// TwinCAT 3 PLC project shelf
// Title: Shelf
// Company: Stefan Lehmann
// ProjectVersion: 0.0.1
// ProgramVersion: 3.1.4026.14
// libraries:
//   Shelf, * (Stefan Lehmann)
//   Tc2_System, * (Beckhoff Automation GmbH)
//   Tc2_Utilities, * (Beckhoff Automation GmbH)
//   Tc3_Module, * (Beckhoff Automation GmbH)
// project tree:
//   / ClassDiagram.TcCD (not stored), PlcTask.TcTTO
//   classes/ FifoBuffer.TcPOU, FlexiBuffer.TcPOU, Part.TcPOU, Shelf.TcPOU, ShelfElement.TcPOU
//   enums/ MainState.TcDUT, TestFlexiBufferState.TcDUT
//   interfaces/ IPart.TcIO, IShelf.TcIO, IShelfElement.TcIO
//   programs/ main.TcPOU
//   programs/tests/ testFlexiBuffer.TcPOU, testShelf.TcPOU
// real-time tasks:
//   TASK PlcTask: cycle T#10ms, priority 1, ADS port 350
//   TASK Standard: cycle T#10ms, priority 20, ADS port 351

CONFIGURATION shelf
    RESOURCE PLC ON TwinCAT3
        TASK PlcTask(INTERVAL := T#10ms, PRIORITY := 1);
        PROGRAM main WITH PlcTask : main;
    END_RESOURCE
END_CONFIGURATION

// ---- enums/MainState.TcDUT
{attribute 'qualified_only'}
{attribute 'strict'}
{attribute 'to_string'}
TYPE MainState :
(
	INIT,
	WAIT,
	ADD_PART1,
	ADD_PART2,
	GET_NEXT_FREE_SHELF_SPACE,
	GET_NEXT_OCCUPIED_SHELF_SPACE,
	GET_SHELF_SPACE_BY_PARTID,
	UNLOAD_NEXT_OCCUPIED_SHELF_SPACE,
	UNLOAD_PART_BY_ID,
	STORE_PART_BY_ROW_COLUMN,
	UNLOAD_PART_BY_ROW_COLUMN
);
END_TYPE

// ---- enums/TestFlexiBufferState.TcDUT
{attribute 'qualified_only'}
{attribute 'strict'}
{attribute 'to_string'}
TYPE TestFlexiBufferState :
(
	INIT,
	ADD_ELEMENT,
	REMOVE_ELEMENT,
	WAIT
);
END_TYPE

// ---- interfaces/IPart.TcIO
INTERFACE IPart EXTENDS __SYSTEM.IQueryInterface

PROPERTY id : String(23)
GET
END_GET
END_PROPERTY

END_INTERFACE

// ---- interfaces/IShelf.TcIO
INTERFACE IShelf EXTENDS __SYSTEM.IQueryInterface

METHOD getNextFreeSpace : IShelfElement
VAR_INPUT
END_VAR
END_METHOD

METHOD getNextOccupiedSpace : IShelfElement
VAR_INPUT
END_VAR
END_METHOD

METHOD getShelfSpaceByPartId : IShelfElement
VAR_INPUT
	partId: STRING(23);
END_VAR
END_METHOD

PROPERTY m : UINT
GET
END_GET
END_PROPERTY

PROPERTY n : UINT
GET
END_GET
END_PROPERTY

METHOD storeNextPart : BOOL
VAR_INPUT
	part: IPart;
END_VAR
END_METHOD

METHOD storePartByRowColumn : IShelfElement
VAR_INPUT
	part: IPart;
	row: UINT;
	column: UINT;
END_VAR
END_METHOD

METHOD unloadNextPart : IPart
VAR_INPUT
END_VAR
END_METHOD

METHOD unloadPartById : IPart
VAR_INPUT
	partId: STRING(23);
END_VAR
END_METHOD

METHOD unloadPartByRowColumn : IPart
VAR_INPUT
	row: UINT;
	column: UINT;
END_VAR
END_METHOD

END_INTERFACE

// ---- interfaces/IShelfElement.TcIO
INTERFACE IShelfElement EXTENDS __System.IQueryInterface

PROPERTY column : UINT
GET
END_GET
SET
END_SET
END_PROPERTY

PROPERTY isOccupied : BOOL
GET
END_GET
END_PROPERTY

PROPERTY part : IPart
GET
END_GET
END_PROPERTY

PROPERTY row : UINT
GET
END_GET
SET
END_SET
END_PROPERTY

METHOD store : BOOL
VAR_INPUT
	part: IPart;
END_VAR
END_METHOD

METHOD unload : IPart
VAR_INPUT
END_VAR
END_METHOD

END_INTERFACE

// ---- programs/main.TcPOU
PROGRAM main
VAR
END_VAR

// Main function for testing some functionality

testShelf();

// testFlexiBuffer();

END_PROGRAM

// ---- programs/tests/testShelf.TcPOU
PROGRAM testShelf
VAR
	shelf: Shelf(2, 2);
	part1: Part('part1');
	part2: Part('part2');
	
	shelfElement: IShelfElement;
	part: IPart;
	
	unloadPartById: BOOL;
	state: MainState;
END_VAR

CASE state OF
MainState.INIT:
	;

// add parts
MainState.ADD_PART1:
	shelf.storeNextPart(part1);
	
MainState.ADD_PART2:
	shelf.storeNextPart(part2);
	
// get spaces
MainState.GET_NEXT_FREE_SHELF_SPACE:
	shelfElement := shelf.getNextFreeSpace();

MainState.GET_NEXT_OCCUPIED_SHELF_SPACE:
	shelfElement := shelf.getNextOccupiedSpace();

MainState.GET_SHELF_SPACE_BY_PARTID:
	shelfElement := shelf.getShelfSpaceByPartId('part2');

// unload parts	
MainState.UNLOAD_NEXT_OCCUPIED_SHELF_SPACE:
	part := shelf.unloadNextPart();

MainState.UNLOAD_PART_BY_ID:
	part := shelf.unloadPartById('part2');
	
// inventory methods
MainState.STORE_PART_BY_ROW_COLUMN:
	shelf.storePartByRowColumn(part1, 1, 1);
	
MainState.UNLOAD_PART_BY_ROW_COLUMN:
	part := shelf.unloadPartByRowColumn( 1, 1);
END_CASE

state := MainState.WAIT;

END_PROGRAM

// ---- classes/Shelf.TcPOU
FUNCTION_BLOCK Shelf IMPLEMENTS IShelf
VAR_INPUT
END_VAR
VAR_OUTPUT
END_VAR
VAR
	rowCount : UINT;
   	columnCount : UINT;
	spaces: ARRAY[0..MAX_ROWS, 0..MAX_COLUMNS] OF ShelfElement();
	freeSpaces: FlexiBuffer;
	occupiedSpaces: FlexiBuffer;
END_VAR
VAR CONSTANT
	MAX_COLUMNS: INT := 1;
	MAX_ROWS: INT := 1;
END_VAR

//FB_Init is always available implicitly and it is used primarily for initialization.
//The return value is not evaluated. For a specific influence, you can also declare the
//methods explicitly and provide additional code there with the standard initialization
//code. You can evaluate the return value.
METHOD FB_Init: BOOL
VAR_INPUT
    bInitRetains: BOOL; // TRUE: the retain variables are initialized (reset warm / reset cold)
    bInCopyCode: BOOL;  // TRUE: the instance will be copied to the copy code afterward (online change)   
	nRows: UINT := 10;
	mColumns: UINT := 10;
END_VAR
VAR
	i: UINT;
	j: UINT;
	k: UINT := 0;
	shelfElement: IShelfElement;
END_VAR
THIS^.rowCount := nRows;
THIS^.columnCount := mColumns;

FOR i:=0 TO nRows - 1 DO
	FOR j:=0 TO mColumns - 1 DO
		shelfElement := THIS^.spaces[i, j];
		shelfElement.row := i;
		shelfElement.column := j;
		THIS^.freeSpaces.addElement(shelfElement); 
	END_FOR
END_FOR
END_METHOD

{warning 'Methodenimplementierung hinzufügen'}
METHOD getNextFreeSpace : IShelfElement
VAR
	freeShelfElement: IShelfElement;
END_VAR
getNextFreeSpace := THIS^.freeSpaces.getFirstElement();
END_METHOD

{warning 'Methodenimplementierung hinzufügen'}
METHOD getNextOccupiedSpace : IShelfElement
VAR
	occupiedShelfElement: IShelfElement;
END_VAR
getNextOccupiedSpace := THIS^.occupiedSpaces.getFirstElement();
END_METHOD

{warning 'Methodenimplementierung hinzufügen'}
METHOD getShelfSpaceByPartId : IShelfElement
VAR_INPUT
	partId: String(23);
END_VAR
VAR
	i: UINT;
	j: UINT;
	shelfElement: IShelfElement;
END_VAR
FOR i:=0 TO THIS^.rowCount - 1 DO
	FOR j:=0 TO THIS^.columnCount - 1 DO
		shelfElement := THIS^.spaces[i, j];
		IF NOT(shelfElement.part = 0) THEN
			IF shelfElement.part.id = partId THEN
				getShelfSpaceByPartId := shelfElement;
				RETURN;
			END_IF;
		END_IF
	END_FOR
END_FOR
END_METHOD

{warning 'Add property implementation'}
PROPERTY m : UINT
GET
m := THIS^.columnCount;
END_GET
END_PROPERTY

{warning 'Add property implementation'}
PROPERTY n : UINT
GET
n := THIS^.rowCount;
END_GET
END_PROPERTY

METHOD storeNextPart : BOOL
VAR_INPUT
	part: IPart;
END_VAR
VAR
	shelfElement: IShelfElement;
END_VAR
shelfElement := THIS^.freeSpaces.removeFirstElement();
IF NOT (shelfElement = 0) THEN
	shelfElement.store(part);
	THIS^.occupiedSpaces.addElement(shelfElement);
END_IF
END_METHOD

{warning 'Add method implementation '}
METHOD storePartByRowColumn : IShelfElement
VAR_INPUT
	part: IPart;
	row	: UINT;
	column	: UINT;
END_VAR
VAR
	shelfElement: IShelfElement;
END_VAR
shelfElement := THIS^.spaces[row, column];

shelfElement.store(part);

IF NOT shelfElement.isOccupied THEN
	THIS^.freeSpaces.removeElement(shelfElement);
	THIS^.occupiedSpaces.addElement(shelfElement);
END_IF;
END_METHOD

{warning 'Methodenimplementierung hinzufügen'}
METHOD unloadNextPart : IPart
VAR
	shelfElement: IShelfElement;
END_VAR
// remove element from occupied spaces
shelfElement := THIS^.occupiedSpaces.removeFirstElement();

IF NOT(shelfElement=0) THEN
	// store part and set to 0
	unloadNextPart := shelfElement.unload();
	// add to free spaces
	THIS^.freeSpaces.addElement(shelfElement);
END_IF;
END_METHOD

{warning 'Methodenimplementierung hinzufügen'}
METHOD unloadPartById : IPart
VAR_INPUT
	partId: STRING(23);
END_VAR
VAR
	shelfElement: IShelfElement;
	part: IPart;
END_VAR
shelfElement := THIS^.getShelfSpaceByPartId(partId);
IF NOT(shelfElement = 0) THEN
	THIS^.occupiedSpaces.removeElement(shelfElement);
	THIS^.freeSpaces.addElement(shelfElement);
	unloadPartById := shelfElement.unload();
END_IF
END_METHOD

{warning 'Add method implementation '}
METHOD unloadPartByRowColumn : IPart
VAR_INPUT
	row	: UINT;
	column	: UINT;
END_VAR
VAR
	shelfElement: IShelfElement;
	part: IPart;
END_VAR
shelfElement := THIS^.spaces[row, column];
IF shelfElement.isOccupied THEN
	part := shelfElement.unload();
	THIS^.freeSpaces.addElement(shelfElement);
	THIS^.occupiedSpaces.removeElement(shelfElement);
END_IF

unloadPartByRowColumn := part;
END_METHOD

END_FUNCTION_BLOCK

// ---- classes/ShelfElement.TcPOU
FUNCTION_BLOCK ShelfElement IMPLEMENTS IShelfElement
VAR_INPUT
END_VAR
VAR_OUTPUT
END_VAR
VAR
	_column: UINT;
	_row: UINT;
	_part: IPart;
	_isOccupied: BOOL := FALSE;
END_VAR
VAR CONSTANT
	ID_SIZE: INT := 23;
END_VAR

{warning 'Add property implementation'}
PROPERTY column : UINT
GET
column := THIS^._column;
END_GET
SET
THIS^._column := column;
END_SET
END_PROPERTY

{warning 'Add property implementation'}
PROPERTY isOccupied : BOOL
GET
isOccupied := THIS^._isOccupied;
END_GET
END_PROPERTY

PROPERTY part : IPart
GET
part := THIS^._part;
END_GET
END_PROPERTY

{warning 'Add property implementation'}
PROPERTY row : UINT
GET
row := THIS^._row;
END_GET
SET
THIS^._row := row;
END_SET
END_PROPERTY

METHOD store : BOOL
VAR_INPUT
	part: IPart;
END_VAR
THIS^._part := part;
THIS^._isOccupied := TRUE;
END_METHOD

METHOD unload : IPart
VAR_INPUT
END_VAR
unload := THIS^.part;
THIS^._part := 0;
THIS^._isOccupied := FALSE;
END_METHOD

END_FUNCTION_BLOCK

// ---- classes/Part.TcPOU
FUNCTION_BLOCK Part IMPLEMENTS IPart
VAR_INPUT
END_VAR
VAR_OUTPUT
END_VAR
VAR
	_id: STRING(23);
END_VAR

//FB_Init is always available implicitly and it is used primarily for initialization.
//The return value is not evaluated. For a specific influence, you can also declare the
//methods explicitly and provide additional code there with the standard initialization
//code. You can evaluate the return value.
METHOD FB_Init: BOOL
VAR_INPUT
    bInitRetains: BOOL; // TRUE: the retain variables are initialized (reset warm / reset cold)
    bInCopyCode: BOOL;  // TRUE: the instance will be copied to the copy code afterward (online change)
	id: String(23);   
END_VAR
THIS^._id := id;
END_METHOD

{warning 'Eigenschaftenimplementierung hinzufügen'}
PROPERTY id : STRING(23)
GET
id := THIS^._id;
END_GET
SET
THIS^._id := id;
END_SET
END_PROPERTY

END_FUNCTION_BLOCK

// ---- classes/FlexiBuffer.TcPOU
FUNCTION_BLOCK FlexiBuffer
VAR_INPUT
END_VAR
VAR_OUTPUT
END_VAR
VAR
	buffer: ARRAY[0..MAX_BUFFER_SIZE - 1] OF IShelfElement;
	count: UINT := 0;
END_VAR
VAR CONSTANT
	MAX_BUFFER_SIZE : UINT := 4;
END_VAR

METHOD addElement : BOOL
VAR_INPUT
	shelfElement: IShelfElement;
END_VAR
THIS^.buffer[THIS^.count] := shelfElement;
THIS^.count := THIS^.count + 1;
END_METHOD

METHOD getFirstElement : IShelfElement
VAR_INPUT
END_VAR
IF count > 0 THEN
	getFirstElement := THIS^.buffer[0];
END_IF;
END_METHOD

METHOD removeElement : BOOL
VAR_INPUT
	shelfElement: IShelfElement;
END_VAR

VAR
	i: UINT;
	j: UINT;
END_VAR
// move elements left in the array
IF THIS^.count > 0 THEN
	FOR i:=0 TO THIS^.count - 1 DO
		IF THIS^.buffer[i] = shelfElement THEN
//			// slower: using for loop		
//  		FOR j:=i+1 TO THIS^.count -1 DO
//  			THIS^.buffer[j-1] := THIS^.buffer[j];
//  		END_FOR
			
			// faster: using memmove
			MEMMOVE(ADR(THIS^.buffer[i]), ADR(THIS^.buffer[i+1]), THIS^.count - i);
		END_IF;  
	END_FOR
	count := count - 1;
END_IF;
END_METHOD

METHOD removeFirstElement : IShelfElement
VAR_INPUT
END_VAR
VAR
	i: UINT;
END_VAR
IF THIS^.count > 0 THEN
	removeFirstElement := THIS^.buffer[0];
// 	// slower: using for loop
// 	FOR i:=1 TO THIS^.COUNT - 1 DO
// 		THIS^.buffer[i-1] := THIS^.buffer[i]; 
// 	END_FOR
	
	// faster: memmove
	MEMMOVE(ADR(THIS^.buffer[0]), ADR(THIS^.buffer[1]), THIS^.count - 1);
	THIS^.count := THIS^.count - 1;
END_IF;
END_METHOD

END_FUNCTION_BLOCK

// ---- classes/FifoBuffer.TcPOU
FUNCTION_BLOCK FifoBuffer
VAR_INPUT
	bOverwrite	: BOOL;
	in 			: IShelfElement;
END_VAR
VAR_OUTPUT
	bOk			: BOOL;
	nCount		: UDINT;
	nLoad		: UDINT;
	out			: IShelfElement;
END_VAR
VAR
	arrBuffer 	: ARRAY[0..MAX_BUFFER_SIZE] OF BYTE; (* Buffer memory used by FB_MemRingBuffer function block *)
	fbBuffer	: FB_MemRingBuffer;
END_VAR
VAR CONSTANT
	MAX_BUFFER_SIZE : UDINT := 1000;
END_VAR

;

ACTION A_Add:
fbBuffer.A_AddTail( pWrite:= ADR( in ),
					cbWrite:= SIZEOF( in ),
					pBuffer:= ADR( arrBuffer ),
					cbBuffer:= SIZEOF( arrBuffer ),
					bOk=> bOk,
					nCount => nCount );


IF NOT bOk THEN (* overflow ? *)
	IF bOverwrite THEN
		fbBuffer.A_RemoveHead(); (* remove one oldest entry *)

		fbBuffer.A_AddTail( bOk => bOk, nCount => nCount );
	END_IF
END_IF



nLoad := (fbBuffer.cbSize * 100) / MAX_BUFFER_SIZE;
END_ACTION

ACTION A_Get:
fbBuffer.A_GetHead( pRead:= ADR( out ),
					cbRead:= SIZEOF( out ),
					pBuffer:= ADR( arrBuffer ),
					cbBuffer:= SIZEOF( arrBuffer ),
					bOk=> bOk,
					nCount => nCount );

nLoad := (fbBuffer.cbSize * 100) / MAX_BUFFER_SIZE;
END_ACTION

ACTION A_Remove:
fbBuffer.A_RemoveHead( 	pRead:= ADR( out ),
						cbRead:= SIZEOF( out ),
						pBuffer:= ADR( arrBuffer ),
						cbBuffer:= SIZEOF( arrBuffer ),
						bOk=> bOk,
						nCount => nCount );

nLoad := (fbBuffer.cbSize * 100) / MAX_BUFFER_SIZE;
END_ACTION

ACTION A_Reset:
MEMSET( ADR( arrBuffer ), 0, SIZEOF( arrBuffer ) ); (* reset (optional) internal buffer *)

fbBuffer.A_Reset( 	bOk=> bOk,
					nCount => nCount );

nLoad := (fbBuffer.cbSize * 100) / MAX_BUFFER_SIZE;
END_ACTION

END_FUNCTION_BLOCK

// ---- programs/tests/testFlexiBuffer.TcPOU
PROGRAM testFlexiBuffer
VAR
	shelf : Shelf(2, 2);
	shelfElements: ARRAY[0..100] OF ShelfElement;
	
	flexibuf: FlexiBuffer;
	state: TestFlexiBufferState;
	
	shelfElement: IShelfElement;
	
	usedElementsCount: UINT := 0;
	i: UINT;
END_VAR


shelf.getNextFreeSpace();

CASE state OF
TestFlexiBufferState.INIT:
	FOR i:=0 TO 3 DO
		usedElementsCount := usedElementsCount + 1;
		flexibuf.addElement(shelfElements[usedElementsCount - 1]);
	END_FOR;
	state := TestFlexiBufferState.WAIT;
	
TestFlexiBufferState.ADD_ELEMENT:
	usedElementsCount := usedElementsCount + 1;	
	flexibuf.addElement(shelfElements[usedElementsCount-1]);	
	state := TestFlexiBufferState.WAIT;

TestFlexiBufferState.REMOVE_ELEMENT:
	shelfElement := flexibuf.removeFirstElement();
	state := TestFlexiBufferState.WAIT;
	
END_CASE

END_PROGRAM
